FUNCTION_BLOCK Resetting IMPLEMENTS ITF_PackMLState, ITF_States
VAR
	_MyContext : ITF_PackMLMachine;
	_MyNextState : ITF_PackMLState;
	_MyStoppingState : ITF_PackMLState;
	_MyAbortingState : ITF_PackMLState;
	_MyName : STRING(20) := 'Resetting';
END_VAR

PROPERTY AbortingState : ITF_PackMLState
GET
AbortingState := _MyAbortingState;
END_GET
SET
_MyAbortingState := AbortingState;
END_SET
END_PROPERTY

METHOD CyclicLogic : BOOL
VAR_INPUT
END_VAR
_MyContext.ChangeState(MyNextState);
END_METHOD

{warning 'add method implementation '}
METHOD EStop : BOOL
END_METHOD

{warning 'add property implementation'}
PROPERTY MyNextState : ITF_PackMLState
GET
MyNextState := _MyNextState;
END_GET
SET
_MyNextState := MyNextState;
END_SET
END_PROPERTY

PROPERTY MyStateName : String(20)
GET
MyStateName := _MyName;
END_GET
END_PROPERTY

{warning 'add method implementation '}
METHOD Reset : BOOL
END_METHOD

METHOD SetContext : BOOL
VAR_INPUT
	context	: ITF_PackMLMachine;
END_VAR
_MyContext := context;
END_METHOD

{warning 'add method implementation '}
METHOD Start : BOOL
END_METHOD

{warning 'add method implementation '}
METHOD Stop : BOOL
END_METHOD

{warning 'add property implementation'}
PROPERTY StoppingState : ITF_PackMLState
GET
StoppingState := _MyStoppingState;
END_GET
SET
_MyStoppingState := StoppingState;
END_SET
END_PROPERTY

END_FUNCTION_BLOCK

(* stored: Version 1.1.0.1, ProductVersion 3.1.4024.12
   POU Resetting: Id {a04f2b88-54e0-4f9d-96c2-2413b8f8730d}, SpecialFunc None
   Property AbortingState: Id {5744e6fe-0ccf-422c-951d-84cd9c9ddf9b}
   Get Get: Id {89625353-a5c6-4769-ace3-c8ff7d78ba97}
   Set Set: Id {7282a72e-f535-497a-903e-017c4f3e493f}
   Method CyclicLogic: Id {3fe49579-6c57-41a1-89d6-f13a605f4ed3}
   Method EStop: Id {78564e11-a330-4481-9f40-b5bfe72c172c}
   Property MyNextState: Id {7172bab1-6091-4f50-a933-5cc3a2c680ff}
   Get Get: Id {2d2f6e95-8816-49a1-865c-e99122bb1747}
   Set Set: Id {4e974532-2531-492d-85e8-b4f190a334a5}
   Property MyStateName: Id {2e035ead-7d36-4408-95bb-61ded047f91d}
   Get Get: Id {ae567aa1-f38e-49db-af2b-df964634d7f4}
   Method Reset: Id {3eeefcff-7251-4a92-9417-b79f79efa8cc}
   Method SetContext: Id {f22654db-fe71-4a75-9e91-cbb3916e52e5}
   Method Start: Id {43d98a02-e31f-4f4c-a038-9348e3d08df8}
   Method Stop: Id {349ec728-9daf-4fbf-b132-65798d14f7a9}
   Property StoppingState: Id {0f308e6f-b249-4db4-80ff-9b59137dd4a7}
   Get Get: Id {75a8732a-d0ed-420f-a152-750d83266cd0}
   Set Set: Id {88e920f6-ce9d-4794-a6d1-8191625a44a8} *)
